RoboDK station: WeldingStation.rdk

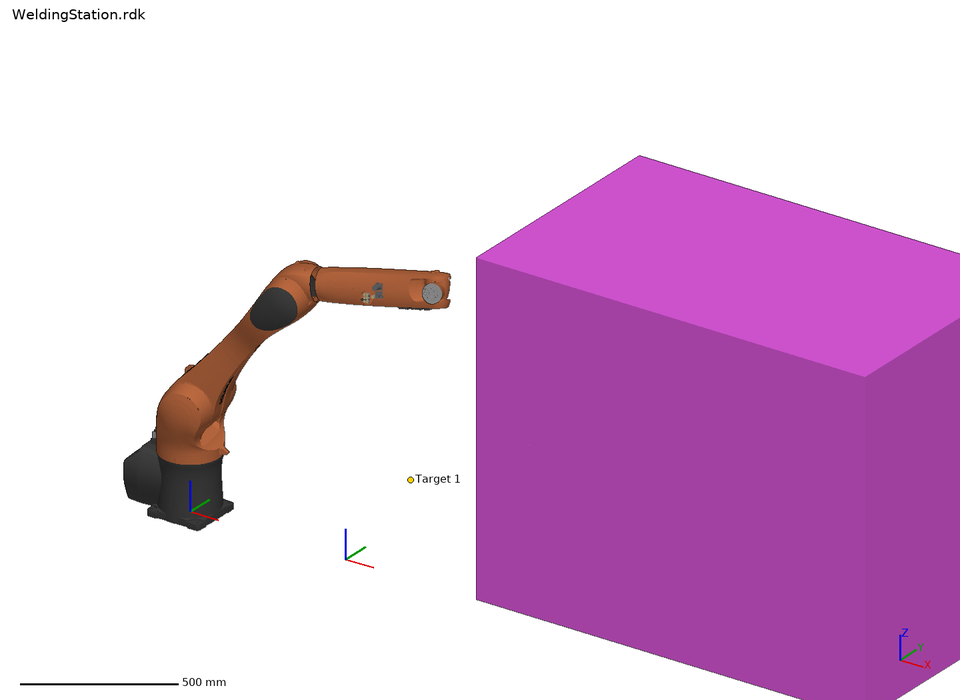
[picture v0: the station drawn from its stored meshes, robots at their saved joint values, targets as dots, program paths as lines]
Station WeldingStation (saved by RoboDK 6.0.4). Poses are relative to the parent item; angles as X-Y-Z fixed-axis rotations.
  - frame KUKA KR 10 R1100 sixx Base at (0, 0, 0) mm
    - robot KUKA KR 10 R1100 sixx: 6 axes, payload 10 kg, reach 1101 mm, repeatability 0.03 mm, weight 54 kg
        modified DH rows (alpha deg, a mm, theta deg, d mm): 0, 0, 0, 400; -90, 25, 0, 0; 0, 560, -90, 0; -90, 35, 0, 515; 90, 0, 0, 0; -90, 0, 180, 80
        joint limits [-170, -190, -120, -185, -120, -350] to [170, 45, 156, 185, 120, 350]; home [0, -90, 90, 0, 0, 0]; saved at [-9.22, -52.82, 43.64, -75.54, -75.91, 45.25]
      - tool WeldingTorch, TCP at (0, 0, 100) mm
  - frame WorkpieceFrame at (600, 0, 0) mm
    - object Workpiece at (500, 0, 0) mm, size 1500 x 900 x 1200 mm, geometry from 01_box_box_flat_touching.step
    - target Target 1 (Cartesian target) at (250, 0, 350) mm, rotated rx 0 ry 0 rz 180 deg; joints [-54.118, 28.976, 39.835, -54.193, -106.119, -19.9] of KUKA KR 10 R1100 sixx
  - program Prog1 (3 instructions, listed below)

--- program Prog1 (robot KUKA KR 10 R1100 sixx) ---
  Set Ref.: WorkpieceFrame
  Set Tool: WeldingTorch
  MoveJ (Target 1)
